(* PLC project AlarmHandlerTemplate, Industrial AI Agent CODESYS 3.5.21.0 *)
(* stored: creationDateTime 2026-06-10T10:00:00, modificationDateTime 2026-06-10T10:00:00 *)

FUNCTION_BLOCK FB_AlarmHandler
  VAR_INPUT
    xTrigger : BOOL;  (* Alarm tetikleme kosulu (TRUE = alarm var) *)
    xAcknowledge : BOOL;  (* Operator kabul (acknowledge) butonu *)
    bLevel : USINT;  (* Alarm seviyesi (0=info, 1=uyari, 2=kritik) *)
  END_VAR
  VAR_OUTPUT
    xActive : BOOL;  (* Alarm kosulu su an aktif mi *)
    xLatched : BOOL;  (* Mandalli alarm: tetiklendi, henuz kabul edilmedi *)
    xUnacknowledged : BOOL;  (* Aktif/mandalli ve kabul bekliyor (yanip sonme icin) *)
    bAlarmLevel : USINT;  (* Mandallanan alarmin seviyesi *)
  END_VAR
  VAR
    rtrigTrigger : R_TRIG;
    rtrigAck : R_TRIG;
  END_VAR

                        
// ------------------------------------------------------------
// FB_AlarmHandler - Alarm mandalla / kabul mantigi
// Tetikleme yukselen kenarda alarmi mandalar ve seviyesini saklar.
// Kabul (acknowledge) yalnizca kosul dustukten sonra mandali siler.
// ------------------------------------------------------------

// Kenar tespiti
rtrigTrigger(CLK := xTrigger);
rtrigAck(CLK := xAcknowledge);

// Anlik aktif durum
xActive := xTrigger;

// --- Mandalla: yukselen kenarda alarmi yakala ve seviye sakla ---
IF rtrigTrigger.Q THEN
    xLatched := TRUE;
    bAlarmLevel := bLevel;
END_IF

// --- Kabul: yalnizca kosul artik aktif degilse mandali sil ---
IF rtrigAck.Q AND NOT xActive THEN
    xLatched := FALSE;
    bAlarmLevel := 0;
END_IF

// --- Kabul bekleyen (yanip sonen) durum ---
// Aktif veya mandalli ise ve henuz temizlenmemisse kabul bekliyor
xUnacknowledged := xActive OR xLatched;

                    
END_FUNCTION_BLOCK
